{attribute 'linkalways'} 
{attribute 'no_explicit_call' := 'This FB is a CLASS and must be accessed using methods or properties'}
{attribute 'enable_dynamic_creation'}
FUNCTION_BLOCK Node_F_VN_ContourOrientationExp EXTENDS VisionNode
VAR
    ipContour : _ITcVnContainer;
    stOrientation : _TcVnRotatedRectangle;
    eMethod : _ETcVnOrientationMethod(ETcVnOrientationMethod.TCVN_OM_PCA);
    hrPrev : _HRESULT(S_OK);
	hresult : _HRESULT(S_OK);
END_VAR

METHOD PUBLIC  Clone : I_Node
VAR
	pNode : POINTER TO Node_F_VN_ContourOrientationExp;
END_VAR
pNode := __NEW(Node_F_VN_ContourOrientationExp);
Clone := pNode^;
END_METHOD

METHOD FB_init : BOOL
VAR_INPUT
	bInitRetains : BOOL; // if TRUE, the retain variables are initialized (warm start / cold start)
	bInCopyCode : BOOL;  // if TRUE, the instance afterwards gets moved into the copy code (online change)
END_VAR
AddInput('ipContour', ipContour);
AddParameter('eMethod', eMethod);
AddInput('hrPrev', hrPrev);
AddOutput('stOrientation', stOrientation);
AddOutput('hresult',hresult);
END_METHOD

METHOD PROTECTED OnExecute
hresult.Value := F_VN_ContourOrientationExp(
	ipContour := ipContour.Value,
    stOrientation := stOrientation.Value,
    eMethod := eMethod.Value,
	hrPrev:= hrPrev.Value);
END_METHOD

METHOD PUBLIC PreExecutionCheck
VAR_INPUT
	Check : I_PreExecutionChecks;
END_VAR
Check.IsTrue((ipContour.IsType(TC_GLOBAL_CONST_LIST.ContainerType_Vector_TcVnPoint2_DINT) OR
              ipContour.IsType(TC_GLOBAL_CONST_LIST.ContainerType_Vector_TcVnPoint2_REAL) OR
              ipContour.IsType(TC_GLOBAL_CONST_LIST.ContainerType_Vector_TcVnPoint2_LREAL)),
              'ipContour contains incorrect type');
END_METHOD

END_FUNCTION_BLOCK

(* stored: Version 1.1.0.1, ProductVersion 3.1.4026.13
   POU Node_F_VN_ContourOrientationExp: Id {3ab382dc-b8f0-0a7f-397c-315ceabf30c6}, SpecialFunc None
   Folder Constructor: Id {b4e8b06f-e2c8-092b-1b51-531847370156}
   Method Clone: Id {8f5831f4-fae1-0533-3867-085f80ad2a0e}
   Method FB_init: Id {13517210-2414-0e65-1b4f-aaa5e236e43a}
   Method OnExecute: Id {78a40f01-c20d-0898-139e-26fd41cc2253}
   Method PreExecutionCheck: Id {f9e18d6f-7618-03e1-3e58-fb9a535315e9} *)
